// Mitsubishi GX Works2 project: Servo_Chay_Nhieu_Vi_Tri   PLC: FX3U/FX3UC

PROGRAM MAIN
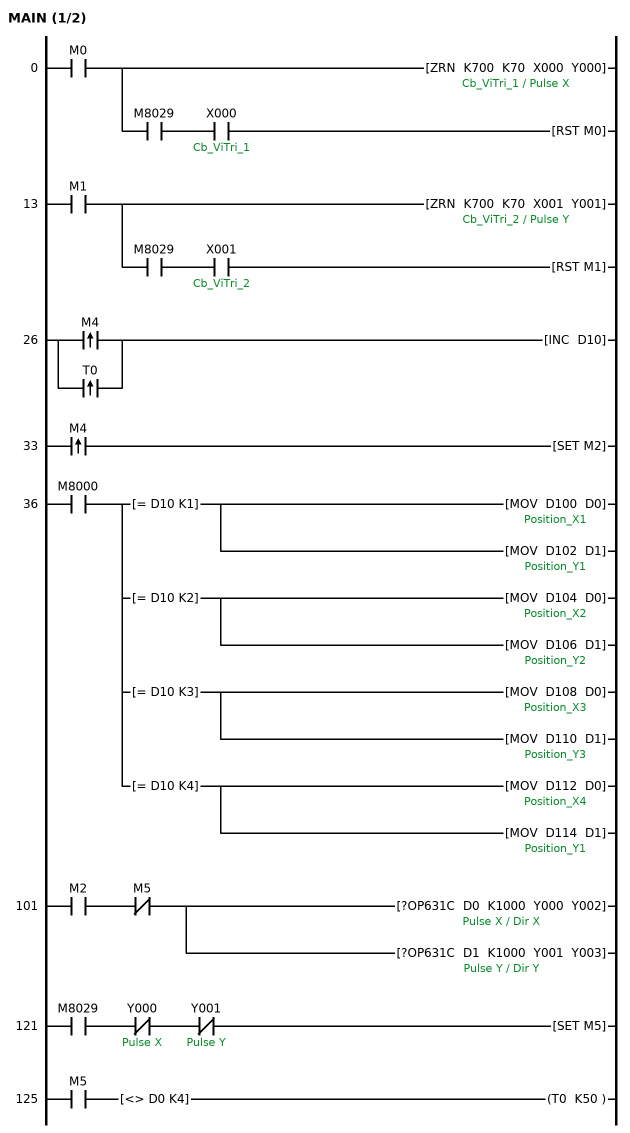
0     LD      M0
      ZRN     K700 K70 X000 Y000  ; Cb_ViTri_1 / Pulse X
      AND     M8029
      AND     X000  ; Cb_ViTri_1
      RST     M0
13    LD      M1
      ZRN     K700 K70 X001 Y001  ; Cb_ViTri_2 / Pulse Y
      AND     M8029
      AND     X001  ; Cb_ViTri_2
      RST     M1
26    LDP     M4
      ORP     T0
      INC     D10
33    LDP     M4
      SET     M2
36    LD      M8000
      MPS
      AND=    D10 K1
      MOV     D100 D0  ; Position_X1
      MOV     D102 D1  ; Position_Y1
      MRD
      AND=    D10 K2
      MOV     D104 D0  ; Position_X2
      MOV     D106 D1  ; Position_Y2
      MRD
      AND=    D10 K3
      MOV     D108 D0  ; Position_X3
      MOV     D110 D1  ; Position_Y3
      MPP
      AND=    D10 K4
      MOV     D112 D0  ; Position_X4
      MOV     D114 D1  ; Position_Y1
101   LD      M2
      ANI     M5
      ?OP631C D0 K1000 Y000 Y002  ; Dir X
      ?OP631C D1 K1000 Y001 Y003  ; Dir Y
121   LD      M8029
      ANI     Y000  ; Pulse X
      ANI     Y001  ; Pulse Y
      SET     M5
125   LD      M5
      AND<>   D0 K4
      OUT     T0 K50
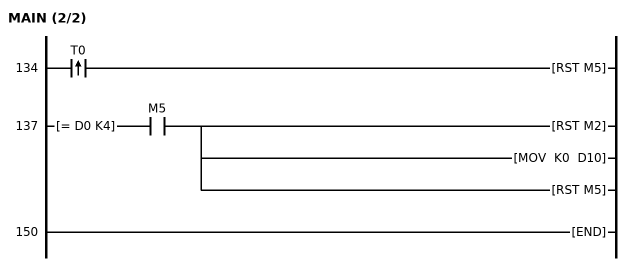
134   LDP     T0
      RST     M5
137   LD=     D0 K4
      AND     M5
      RST     M2
      MOV     K0 D10
      RST     M5
150   END
END_PROGRAM
